// TwinCAT 3 PLC project TcMatrixTest
// Title: TcMatrix Unit Tests
// Company: Burks Engineering
// Author: Andrew Burks
// ProjectVersion: 0.0.0
// Description: Unit Tests for the TcMatrix Library
// ProgramVersion: 3.1.4023.0
// libraries:
//   Tc2_Standard, * (Beckhoff Automation GmbH)
//   Tc2_System, * (Beckhoff Automation GmbH)
//   Tc3_DynamicMemory, * (Beckhoff Automation GmbH)
//   Tc3_Module, * (Beckhoff Automation GmbH)
//   TcMatrix, * (Burks Engineering)
//   TcUnit,1.2.0.0,www.tcunit.org
// project tree:
//   / PlcTask.TcTTO
//   TESTs/ FB_CsvReadWrite_Test.TcPOU, FB_Array_Test.TcPOU, FB_MatrixElementProduct_Test.TcPOU, FB_MatrixDeterminate_Test.TcPOU, FB_MatrixGetMagicSquare_Test.TcPOU, FB_MatrixGrow_Test.TcPOU, FB_MatrixMatrixProduct_Test.TcPOU, FB_MatrixInvert_Test.TcPOU, FB_MatrixShrink_Test.TcPOU, FB_MatrixElementSum_Test.TcPOU, FB_MatrixSubMatrix_Test.TcPOU, FB_DynamicMatrix_Test.TcPOU, FB_MatrixTranspose_Test.TcPOU, FB_StaticMatrix_Test.TcPOU, FB_VectorCrossProduct_Test.TcPOU, PRG_TEST.TcPOU
//   Version/ Global_Version.TcGVL
// real-time tasks:
//   TASK PlcTask: cycle T#10ms, priority 20, ADS port 350

CONFIGURATION TcMatrixTest
    RESOURCE PLC ON TwinCAT3
        TASK PlcTask(INTERVAL := T#10ms, PRIORITY := 20);
        PROGRAM PRG_TEST WITH PlcTask : PRG_TEST;
    END_RESOURCE
END_CONFIGURATION

// ---- Version/Global_Version.TcGVL
{attribute 'TcGenerated'}
{attribute 'no-analysis'}
{attribute 'linkalways'}
// This function has been automatically generated from the project information.
VAR_GLOBAL CONSTANT
	{attribute 'const_non_replaced'}
	stLibVersion_TcMatrix_Unit_Tests : ST_LibVersion := (iMajor := 0, iMinor := 0, iBuild := 0, iRevision := 0, nFlags := 0, sVersion := '0.0.0');
END_VAR

// ---- TESTs/PRG_TEST.TcPOU
PROGRAM PRG_TEST
VAR
	fbDynamicMatrix : FB_DynamicMatrix_Test;
	fbArray: FB_Array_Test;
	fbMatrixGetMagicSquare : FB_MatrixGetMagicSquare_Test;
	fbMatrixSubmatrix : FB_MatrixSubMatrix_Test;
	fbMatrixGrow : FB_MatrixGrow_Test;
	fbMatrixShrink : FB_MatrixShrink_Test;
	fbMatrixElementSum : FB_MatrixElementSum_Test;
	fbMatrixElementProduct : FB_MatrixElementProduct_Test;
	fbMatrixDeterminate : FB_MatrixDeterminate_Test;
	fbMatrixMatrixProduct : FB_MatrixMatrixProduct_Test;
	fbVectorCrossProdcut : FB_VectorCrossProduct_Test;
	fbStaticMatrix : FB_StaticMatrix_Test;
	fbMatrixTranspose : FB_MatrixTranspose_Test;
	fbMatrixInvert : FB_MatrixInvert_Test;
	fbCsvReadWrite : FB_CsvReadWrite_Test;
END_VAR

TcUnit.RUN();

END_PROGRAM

// ---- TESTs/FB_DynamicMatrix_Test.TcPOU
FUNCTION_BLOCK FB_DynamicMatrix_Test EXTENDS FB_TestSuite
VAR_INPUT
END_VAR
VAR_OUTPUT
END_VAR
VAR
END_VAR

WhenInitiallyResizedExpectMemoryAllocated();
WhenResizedBiggerExpectMoreMemoryAllocated();
WhenResizedSmallerExpectLessMemoryAllocated();
WhenResizedToZeroExpectNoMemoryAllocated();

METHOD PRIVATE WhenInitiallyResizedExpectMemoryAllocated
VAR_INPUT
END_VAR

VAR
	M : DynamicMatrix;
	ResizeSuccess : BOOL;

END_VAR
TEST('WhenInitiallyResizedExpectMemoryAllocated');

// @TEST-RUN
ResizeSuccess := M.Resize(1,1,FALSE,TRUE);



// @TEST-ASSERT
AssertTrue(Condition :=ResizeSuccess,
	message := 'Error on valid initial resize');

	
TEST_FINISHED();
END_METHOD

METHOD PRIVATE WhenResizedBiggerExpectMoreMemoryAllocated
VAR_INPUT
END_VAR
VAR
	M : DynamicMatrix;
	InitialResizeSuccess : BOOL;
	SecondResizeSuccess : BOOL;

END_VAR
TEST('WhenResizedBiggerExpectMoreMemoryAllocated');

// @TEST-RUN
InitialResizeSuccess := M.Resize(1,1,FALSE,TRUE);
SecondResizeSuccess := M.Resize(2,2,FALSE,TRUE);


// @TEST-ASSERT
AssertTrue(Condition :=InitialResizeSuccess,
	message := 'Error on valid initial resize');
AssertTrue(Condition :=SecondResizeSuccess,
	message := 'Error on valid second resize');

	
TEST_FINISHED();
END_METHOD

METHOD PRIVATE WhenResizedSmallerExpectLessMemoryAllocated
VAR_INPUT
END_VAR
VAR
	M : DynamicMatrix;
	InitialResizeSuccess : BOOL;
	SecondResizeSuccess : BOOL;
	
END_VAR
TEST('WhenResizedSmallerExpectLessMemoryAllocated');

// @TEST-RUN
InitialResizeSuccess := M.Resize(2,2,FALSE,TRUE);
SecondResizeSuccess := M.Resize(1,1,FALSE,TRUE);

// @TEST-ASSERT
AssertTrue(Condition :=InitialResizeSuccess,
	message := 'Error on valid initial resize');
AssertTrue(Condition :=SecondResizeSuccess,
	message := 'Error on valid second resize');

	
TEST_FINISHED();
END_METHOD

METHOD PRIVATE WhenResizedToZeroExpectNoMemoryAllocated
VAR_INPUT
END_VAR
VAR
	M : DynamicMatrix;
	InitialResizeSuccess : BOOL;
	SecondResizeSuccess : BOOL;

END_VAR
TEST('WhenResizedToZeroExpectNoMemoryAllocated');

// @TEST-RUN
InitialResizeSuccess := M.Resize(1,1,FALSE,TRUE);
SecondResizeSuccess := M.Resize(0,0,FALSE,TRUE);


// @TEST-ASSERT
AssertTrue(Condition :=InitialResizeSuccess,
	message := 'Error on valid initial resize');
AssertTrue(Condition :=SecondResizeSuccess,
	message := 'Error on valid second resize');

	
TEST_FINISHED();
END_METHOD

END_FUNCTION_BLOCK

// ---- TESTs/FB_Array_Test.TcPOU
FUNCTION_BLOCK FB_Array_Test EXTENDS FB_TestSuite
VAR_INPUT
END_VAR
VAR_OUTPUT
END_VAR
VAR
END_VAR

WhenDynamicInitializedExpectValuesCopied();
WhenStaticInitializedExpectValuesCopied();
MarkdownExample1();

METHOD PRIVATE MarkdownExample1
VAR_INPUT
END_VAR
VAR
	M : Array2DStaticMatrix; //This instance is the matrix that the code will interact with
	M_Data : ARRAY[1..3,1..3] OF LREAL; //This array will act as the memory for the matrix
	V : Array2DStaticMatrix; //This instance is the initial column vector
	V_Data : ARRAY[1..3,1..1] OF LREAL := [1, 2, 3]; //This array will act as the memory for the initial column vector, prepopulated
	Res : Array2DStaticMatrix; //This instance is the resulting column vector
	Res_Data : ARRAY[1..3,1..1] OF LREAL := [1, 2, 3]; //This array will act as the memory for the resulting column vector
	success : BOOL; //records success or failure of the matrix multiplication
	equal : BOOL; //records success if the resulting vector is equal to the first
END_VAR
TEST('MarkdownExample1');

// @TEST-RUN
M(Data := M_Data); //Connect the memory to the matrix and initialize it
V(Data := V_Data); //Connect the memory to the initial column vector and initialize it (retaining declared values)
Res(Data := Res_Data); //Connect the memory to the resulting column vector and initialize it

M.FillTrapezoidal(Diagonal := 1, UpperRight := 0, LowerLeft := 0); //Transforms the matrix from all zeros into the identity matrix
success := Matrix_Product(M,V,Res); //perform the matrix multiplication
equal := V.IsEqual(Res); //the result of the multiplication should be equal to the initial value because of the identity matrix
	

// @TEST-ASSERT
AssertTrue(Condition :=success,
	message := 'Error on valid initial resize');
AssertTrue(Condition :=equal,
	message := 'Error on valid initial resize');
TEST_FINISHED();
END_METHOD

METHOD PRIVATE WhenDynamicInitializedExpectValuesCopied
VAR_INPUT
END_VAR
VAR
	A : ARRAY[1..3, 1..3] OF LREAL := [1,2,3,4,5,6,7,8,9];
	M : DynamicMatrix;
	
	InitSuccess : BOOL;
	
	ExpectedRank : UINT := 3;
	ExpectedVal : LREAL := 8.0; //expected at A[3,2] and M(2,1)
	
	MatrixRows : UINT;
	MatrixCols : UINT;
	ArrayVal : LREAL;
	MatrixVal : LREAL;

END_VAR
TEST('WhenDynamicInitializedExpectValuesCopied');

// @TEST-RUN
InitSuccess := M.InitArray2D(A);

MatrixRows := M.Rows;
MatrixCols := M.Cols;
ArrayVal := A[3,2];
MatrixVal := M.GetRC(2,1);


// @TEST-ASSERT
AssertTrue(Condition :=InitSuccess,
	message := 'Error on valid initial resize');
AssertEquals(Expected := ExpectedRank,
	Actual := MatrixRows,
	Message := 'Matrix row size not correct');
AssertEquals(Expected := ExpectedRank,
	Actual := MatrixCols,
	Message := 'Matrix col size not correct');
	
AssertEquals(Expected := ExpectedVal,
	Actual := ArrayVal,
	Message := 'Array content at [3,2] not correct');
	
AssertEquals(Expected := ExpectedVal,
	Actual := MatrixVal,
	Message := 'Matrix content at (2,1) not correct');
	
TEST_FINISHED();
END_METHOD

METHOD PRIVATE WhenStaticInitializedExpectValuesCopied
VAR_INPUT
END_VAR
VAR
	A : ARRAY[1..3, 1..3] OF LREAL := [1,2,3,4,5,6,7,8,9];
	M : Array2DStaticMatrix;
	
	ExpectedRank : UINT := 3;
	ExpectedVal : LREAL := 8.0; //expected at A[3,2] and M(2,1)
	
	MatrixRows : UINT;
	MatrixCols : UINT;
	ArrayVal : LREAL;
	MatrixVal : LREAL;

END_VAR
TEST('WhenStaticInitializedExpectValuesCopied');

// @TEST-RUN
M(Data := A);

MatrixRows := M.Rows;
MatrixCols := M.Cols;
ArrayVal := A[3,2];
MatrixVal := M.GetRC(2,1);


// @TEST-ASSERT
AssertEquals(Expected := ExpectedRank,
	Actual := MatrixRows,
	Message := 'Matrix row size not correct');
AssertEquals(Expected := ExpectedRank,
	Actual := MatrixCols,
	Message := 'Matrix col size not correct');
	
AssertEquals(Expected := ExpectedVal,
	Actual := ArrayVal,
	Message := 'Array content at [3,2] not correct');
	
AssertEquals(Expected := ExpectedVal,
	Actual := MatrixVal,
	Message := 'Matrix content at (2,1) not correct');
	
TEST_FINISHED();
END_METHOD

END_FUNCTION_BLOCK

// ---- TESTs/FB_MatrixGetMagicSquare_Test.TcPOU
FUNCTION_BLOCK FB_MatrixGetMagicSquare_Test EXTENDS FB_TestSuite
VAR_INPUT
END_VAR
VAR_OUTPUT
END_VAR
VAR
END_VAR

WhenCreatedExpectMagicProperties();

METHOD PRIVATE WhenCreatedExpectMagicProperties
VAR_INPUT
END_VAR
VAR
	M1 : DynamicMatrix;
	V : DynamicMatrix;
	Actual : LREAL;
	Expected : LREAL := 15;
	I : UINT;
END_VAR
TEST('WhenCreatedExpectMagicProperties');

// @TEST-RUN
M1.InitMagicSquare(3);//all rows and cols are 15
M1.LogData('3x3 Magic Square');

// @TEST-ASSERT
FOR I := 0 TO M1.Rows-1 DO
	//V.AsRowVector(M1,I); //cannot use, untested at this point
	Actual :=  M1.GetRC(I,0) + M1.GetRC(I,1) + M1.GetRC(I,2);//V.Sum; //cannot use, untested at this point
	AssertEquals(Expected,Actual,'Row is not the magic number');
END_FOR
FOR I := 0 TO M1.Cols-1 DO
	//V.AsRowVector(M1,I); //cannot use, untested at this point
	Actual :=  M1.GetRC(0,I) + M1.GetRC(1,I) + M1.GetRC(2,I);//V.Sum; //cannot use, untested at this point
	AssertEquals(Expected,Actual,'Col is not the magic number');
END_FOR

TEST_FINISHED();
END_METHOD

END_FUNCTION_BLOCK

// ---- TESTs/FB_MatrixSubMatrix_Test.TcPOU
{attribute 'reflection'}
FUNCTION_BLOCK FB_MatrixSubMatrix_Test EXTENDS FB_TestSuite
VAR_INPUT
END_VAR
VAR_OUTPUT
END_VAR
VAR
END_VAR

WhenCreatedExpectDataRetained();

METHOD PRIVATE WhenCreatedExpectDataRetained
VAR_INPUT
END_VAR
VAR
	M1 : DynamicMatrix;
	M2 : DynamicMatrix;
	Result : BOOL;
	
	Ri : UINT;
	Ci : UINT;
	
	Expected : LREAL;
	Actual : LREAL;
END_VAR
TEST('WhenCreatedExpectDataRetained');

// @TEST-RUN
M1.InitMagicSquare(5);
Result := M2.AsSubMatrix(M1,1,3,1,3);

// @TEST-ASSERT
AssertTrue(Result,'Main function call was not successful');

FOR Ri := 0 TO M2.Rows-1 DO
	FOR Ci := 0 TO M2.Cols-1 DO
		Expected := M1.GetRC(Ri+1,Ci+1);
		Actual := M2.GetRC(Ri,Ci);
		AssertEquals(Expected, Actual, 'Equivalent values are not equal after submatrix');
	END_FOR;
END_FOR

TEST_FINISHED();
END_METHOD

END_FUNCTION_BLOCK

// ---- TESTs/FB_MatrixGrow_Test.TcPOU
FUNCTION_BLOCK FB_MatrixGrow_Test EXTENDS FB_TestSuite
VAR_INPUT
END_VAR
VAR_OUTPUT
END_VAR
VAR
END_VAR

WhenEmptyExpectNoError();
WhenGrownExpectDataRetained();
WhenGrownExpectNewDataFilled();

METHOD PRIVATE WhenEmptyExpectNoError
VAR_INPUT
END_VAR
VAR
	M1 : DynamicMatrix;
	M2 : DynamicMatrix;
	Result : BOOL;
END_VAR
TEST('WhenEmptyExpectNoError');

// @TEST-RUN
M1.Init(0,0);
Result := M2.AsGrown(M1,0,0,0,0,0);

// @TEST-ASSERT
AssertTrue(Result,'Main function call was not successful');

TEST_FINISHED();
END_METHOD

METHOD PRIVATE WhenGrownExpectDataRetained
VAR_INPUT
END_VAR
VAR
	M1 : DynamicMatrix;
	M2 : DynamicMatrix;
	M3 : DynamicMatrix;
	Result : BOOL;
END_VAR
TEST('WhenGrownExpectDataRetained');

// @TEST-RUN
M1.InitMagicSquare(3);
Result := M2.AsGrown(M1,0,0,0,0,0);
M3.AsSubMatrix(M2,1,3,1,3);

// @TEST-ASSERT
AssertTrue(Result,'Main function call was not successful');
AssertTrue(M3.IsEqual(M1),'Old data was not retained');

TEST_FINISHED();
END_METHOD

METHOD PRIVATE WhenGrownExpectNewDataFilled
VAR_INPUT
END_VAR
VAR
	M1 : DynamicMatrix;
	M2 : DynamicMatrix;
	Result : BOOL;
END_VAR
TEST('WhenGrownExpectNewDataFilled');

// @TEST-RUN
M1.InitZeros(3,3);
Result := M2.AsGrown(M1,0,0,1,2,3);

// @TEST-ASSERT
AssertTrue(Result,'Main function call was not successful');
AssertTrue(M2.GetRC(0,0) = 1,'Diagonal data was not filled');
AssertTrue(M2.GetRC(0,1) = 2,'Row data was not filled');
AssertTrue(M2.GetRC(1,0) = 3,'Col data was not filled');

TEST_FINISHED();
END_METHOD

END_FUNCTION_BLOCK

// ---- TESTs/FB_MatrixShrink_Test.TcPOU
FUNCTION_BLOCK FB_MatrixShrink_Test EXTENDS FB_TestSuite
VAR_INPUT
END_VAR
VAR_OUTPUT
END_VAR
VAR
END_VAR

WhenEmptyExpectError();
WhenShrunkExpectDataRetained();

METHOD PRIVATE WhenEmptyExpectError
VAR_INPUT
END_VAR
VAR
	M1 : DynamicMatrix;
	M2 : DynamicMatrix;
	Result : BOOL;
END_VAR
TEST('WhenEmptyExpectError');

// @TEST-RUN
M1.InitZeros(1,1);
Result := M2.AsShrunk(M1,0,0);

// @TEST-ASSERT
AssertFalse(Result,'Main function call was unexpectedly successful');

TEST_FINISHED();
END_METHOD

METHOD PRIVATE WhenShrunkExpectDataRetained
VAR_INPUT
END_VAR
VAR
	M1 : DynamicMatrix;
	M2 : DynamicMatrix;
	M3 : DynamicMatrix;
	Result : BOOL;
END_VAR
TEST('WhenShrunkExpectDataRetained');

// @TEST-RUN
M1.InitMagicSquare(3);
Result := M2.AsShrunk(M1,0,0);
M3.AsSubMatrix(M1,1,2,1,2);

// @TEST-ASSERT
AssertTrue(Result,'Main function call was not successful');
AssertTrue(M3.IsEqual(M2),'Old data was not retained');

TEST_FINISHED();
END_METHOD

END_FUNCTION_BLOCK

// ---- TESTs/FB_MatrixElementSum_Test.TcPOU
FUNCTION_BLOCK FB_MatrixElementSum_Test EXTENDS FB_TestSuite
VAR_INPUT
END_VAR
VAR_OUTPUT
END_VAR
VAR
END_VAR

WhenDifferentExpectError();
WhenmatchingExpectResult();

METHOD PRIVATE WhenDifferentExpectError
VAR_INPUT
END_VAR
VAR
	M1 : DynamicMatrix;
	M2 : DynamicMatrix;
	M3 : DynamicMatrix;
	Result : BOOL;
END_VAR
TEST('WhenDifferentExpectError');

// @TEST-RUN
M1.InitMagicSquare(3);
M2.InitMagicSquare(5);
Result := M3.AsElementSum(M1,M2);

// @TEST-ASSERT
AssertFalse(Result,'Main function call was unexpectedly successful');

TEST_FINISHED();
END_METHOD

METHOD PRIVATE WhenMatchingExpectResult
VAR_INPUT
END_VAR
VAR
	M1 : DynamicMatrix;
	M2 : DynamicMatrix;
	M3 : DynamicMatrix;
	Result : BOOL;
END_VAR
TEST('WhenMatchingExpectResult');

// @TEST-RUN
M1.InitMagicSquare(3);
M2.InitMagicSquare(3);
Result := M3.AsElementSum(M1,M2);
M1.Scale(2);

// @TEST-ASSERT
AssertTrue(Result,'Main function call was not successful');
AssertTrue(M3.IsEqual(M1),'Data was successfully added');

TEST_FINISHED();
END_METHOD

END_FUNCTION_BLOCK

// ---- TESTs/FB_MatrixElementProduct_Test.TcPOU
FUNCTION_BLOCK FB_MatrixElementProduct_Test EXTENDS FB_TestSuite
VAR_INPUT
END_VAR
VAR_OUTPUT
END_VAR
VAR
END_VAR

WhenDifferentExpectError();
WhenmatchingExpectResult();

METHOD PRIVATE WhenDifferentExpectError
VAR_INPUT
END_VAR
VAR
	M1 : DynamicMatrix;
	M2 : DynamicMatrix;
	M3 : DynamicMatrix;
	Result : BOOL;
END_VAR
TEST('WhenDifferentExpectError');

// @TEST-RUN
M1.InitMagicSquare(3);
M2.InitMagicSquare(5);
Result := M3.AsElementProduct(M1,M2);

// @TEST-ASSERT
AssertFalse(Result,'Main function call was unexpectedly successful');

TEST_FINISHED();
END_METHOD

METHOD PRIVATE WhenMatchingExpectResult
VAR_INPUT
END_VAR
VAR
	M1 : DynamicMatrix;
	M2 : DynamicMatrix;
	M3 : DynamicMatrix;
	Result : BOOL;
END_VAR
TEST('WhenMatchingExpectResult');

// @TEST-RUN
M1.InitMagicSquare(3);
M2.InitMagicSquare(3);
Result := M3.AsElementProduct(M1,M2);
M1.Power(2);

// @TEST-ASSERT
AssertTrue(Result,'Main function call was not successful');
AssertTrue(M3.IsEqual(M1),'Data was successfully multiplied');

TEST_FINISHED();
END_METHOD

END_FUNCTION_BLOCK

// ---- TESTs/FB_MatrixDeterminate_Test.TcPOU
FUNCTION_BLOCK FB_MatrixDeterminate_Test EXTENDS FB_TestSuite
VAR_INPUT
END_VAR
VAR_OUTPUT
END_VAR
VAR
END_VAR

WhenNotSquareExpectError();
WhenMatchingExpectResult();

METHOD PRIVATE WhenMatchingExpectResult
VAR_INPUT
END_VAR
VAR
	M1 : DynamicMatrix;
	Result : BOOL;
	Actual : LREAL;
	Expected : LREAL := 360;
END_VAR
TEST('WhenMatchingExpectResult');

// @TEST-RUN
M1.InitMagicSquare(3);
Result := Matrix_DeterminateSquare(M := M1,Res => Actual);

// @TEST-ASSERT
AssertTrue(Result,'Main function call was not successful');
AssertEquals(Expected,Actual,'Determinate value was incorrect');

TEST_FINISHED();
END_METHOD

METHOD PRIVATE WhenNotSquareExpectError
VAR_INPUT
END_VAR
VAR
	M1 : DynamicMatrix;
	Result : BOOL;
	Actual : LREAL;
	Expected : LREAL := 0;
END_VAR
TEST('WhenNotSquareExpectError');

// @TEST-RUN
M1.InitTrapezoidal(2,3,1,1,1);
Result := Matrix_DeterminateSquare(M := M1,Res => Actual);

// @TEST-ASSERT
AssertFalse(Result,'Main function call was unexpectedly successful');
AssertEquals(Expected,Actual,'Determinate value was incorrect');

TEST_FINISHED();
END_METHOD

END_FUNCTION_BLOCK

// ---- TESTs/FB_MatrixMatrixProduct_Test.TcPOU
FUNCTION_BLOCK FB_MatrixMatrixProduct_Test EXTENDS FB_TestSuite
VAR_INPUT
END_VAR
VAR_OUTPUT
END_VAR
VAR
END_VAR

WhenColumnsExpectError();
WhenOppositeExpectScalar();
WhenOppositeExpectSquare();
WhenWithIdentityExpectSame();

METHOD PRIVATE WhenColumnsExpectError
VAR_INPUT
END_VAR
VAR
	V1 : DynamicMatrix;
	V2 : DynamicMatrix;
	M1 : DynamicMatrix;
	Result : BOOL;
END_VAR
TEST('WhenColumnsExpectError');

// @TEST-RUN
V1.InitVector(3,1,1);
V2.InitVector(3,1,1);
Result := M1.AsMatrixProduct(V1,V2);

// @TEST-ASSERT
AssertFalse(Result,'Main function call was unexpectedly successful');

TEST_FINISHED();
END_METHOD

METHOD PRIVATE WhenOppositeExpectScalar
VAR_INPUT
END_VAR
VAR
	V1 : DynamicMatrix;
	V2 : DynamicMatrix;
	M1 : DynamicMatrix;
	Result : BOOL;
END_VAR
TEST('WhenOppositeExpectScalar');

// @TEST-RUN
V1.InitVector(3,1,1);
V2.InitVector(3,1,1);
V1.Transpose();
Result := M1.AsMatrixProduct(V1,V2);

// @TEST-ASSERT
AssertTrue(Result,'Main function call was not successful');
AssertTrue(M1.Length = 1,'Result was not a scalar');
AssertTrue(M1.GetI(0) = V1.GetVectorDotProduct(V2),'Result was not the same as a dot product');

TEST_FINISHED();
END_METHOD

METHOD PRIVATE WhenOppositeExpectSquare
VAR_INPUT
END_VAR
VAR
	V1 : DynamicMatrix;
	V2 : DynamicMatrix;
	M1 : DynamicMatrix;
	Result : BOOL;
END_VAR
TEST('WhenOppositeExpectSquare');

// @TEST-RUN
V1.InitVector(3,1,1);
V2.InitVector(3,1,1);
V2.Transpose();
Result := M1.AsMatrixProduct(V1,V2);

// @TEST-ASSERT
AssertTrue(Result,'Main function call was not successful');
AssertTrue(M1.Length = 9 AND M1.IsSquare,'Result was not a 3x3 square');
AssertTrue(M1.Sum = 36,'Result values are incorrect');

TEST_FINISHED();
END_METHOD

METHOD PRIVATE WhenWithIdentityExpectSame
VAR_INPUT
END_VAR
VAR
	V1 : DynamicMatrix;
	MI : DynamicMatrix;
	M1 : DynamicMatrix;
	Result : BOOL;
END_VAR
TEST('WhenWithIdentityExpectSame');

// @TEST-RUN
V1.InitVector(3,1,1);
MI.InitIdentity(3);
Result := M1.AsMatrixProduct(MI,V1);

// @TEST-ASSERT
AssertTrue(Result,'Main function call was not successful');
AssertTrue(V1.IsEqual(M1),'Result was not the same');

TEST_FINISHED();
END_METHOD

END_FUNCTION_BLOCK

// ---- TESTs/FB_VectorCrossProduct_Test.TcPOU
FUNCTION_BLOCK FB_VectorCrossProduct_Test EXTENDS FB_TestSuite
VAR_INPUT
END_VAR
VAR_OUTPUT
END_VAR
VAR
END_VAR

WhenWrongSizeExpectError();
WhenMatchingSizeExpectResult();
WhenBackwardsExpectOppositeResult();

METHOD PRIVATE WhenBackwardsExpectOppositeResult
VAR_INPUT
END_VAR
VAR
	MV : DynamicMatrix;
	V1 : DynamicMatrix;
	V2 : DynamicMatrix;
	V3 : DynamicMatrix;
	Vs : ARRAY[0..1] OF POINTER TO MAtrix;
	M1 : DynamicMatrix;
	Result : BOOL;
END_VAR
TEST('WhenBackwardsExpectOppositeResult');

// @TEST-RUN
Vs[1] := ADR(V1);
Vs[0] := ADR(V2);

MV.InitIdentity(3);
V1.AsColVector(MV,0);
V2.AsColVector(MV,1);
V3.AsColVector(MV,2);
V3.Scale(-1);

Result := M1.AsVectorCrossProduct(Vs);

// @TEST-ASSERT
AssertTrue(Result,'Main function call was not successful');
AssertTrue(M1.IsEqual(V3),'Result is the correct vector');

TEST_FINISHED();
END_METHOD

METHOD PRIVATE WhenMatchingSizeExpectResult
VAR_INPUT
END_VAR
VAR
	MV : DynamicMatrix;
	V1 : DynamicMatrix;
	V2 : DynamicMatrix;
	V3 : DynamicMatrix;
	Vs : ARRAY[0..1] OF POINTER TO MAtrix;
	M1 : DynamicMatrix;
	Result : BOOL;
END_VAR
TEST('WhenMatchingSizeExpectResult');

// @TEST-RUN
Vs[0] := ADR(V1);
Vs[1] := ADR(V2);

MV.InitIdentity(3);
V1.AsColVector(MV,0);
V2.AsColVector(MV,1);
V3.AsColVector(MV,2);

Result := M1.AsVectorCrossProduct(Vs);

// @TEST-ASSERT
AssertTrue(Result,'Main function call was not successful');
AssertTrue(M1.IsEqual(V3),'Result is not the correct vector');

TEST_FINISHED();
END_METHOD

METHOD PRIVATE WhenWrongSizeExpectError
VAR_INPUT
END_VAR
VAR
	V1 : DynamicMatrix;
	V2 : DynamicMatrix;
	Vs : ARRAY [0..1] OF POINTER TO Matrix;
	M1 : DynamicMatrix;
	Result : BOOL;
END_VAR
TEST('WhenWrongSizeExpectError');

// @TEST-RUN
Vs[0] := ADR(V1);
Vs[1] := ADR(V2);

V1.InitVector(3,1,1);
V2.InitVector(4,1,1);

Result := Vector_CrossProduct(M1,Vs);

// @TEST-ASSERT
AssertFalse(Result,'Main function call was unexpectedly successful');

TEST_FINISHED();
END_METHOD

END_FUNCTION_BLOCK

// ---- TESTs/FB_StaticMatrix_Test.TcPOU
FUNCTION_BLOCK FB_StaticMatrix_Test EXTENDS FB_TestSuite
VAR_INPUT
END_VAR
VAR_OUTPUT
END_VAR
VAR
END_VAR

WhenCreatedExpectDataAssignable();

METHOD PRIVATE WhenCreatedExpectDataAssignable
VAR_INPUT
END_VAR
VAR
	M1 : ExternalStaticMatrix;
	M2 : DynamicMatrix;
	Data : ARRAY[0..8] OF LREAL;
	
	
END_VAR
TEST('WhenCreatedExpectDataAssignable');

// @TEST-RUN
M2.InitMagicSquare(3);
M1.Init(ADR(Data),3,3);
M1.FillFrom(M2);


// @TEST-ASSERT
AssertTrue(M1.IsEqual(M2),'Data was not all assigned');

TEST_FINISHED();
END_METHOD

END_FUNCTION_BLOCK

// ---- TESTs/FB_MatrixTranspose_Test.TcPOU
FUNCTION_BLOCK FB_MatrixTranspose_Test EXTENDS FB_TestSuite
VAR_INPUT
END_VAR
VAR_OUTPUT
END_VAR
VAR
END_VAR

WhenSquareExpectTranspose();
WhenDynamicRectangleExpectTranspose();
WhenStaticRectangleExpectTranspose();

METHOD PRIVATE WhenDynamicRectangleExpectTranspose
VAR_INPUT
END_VAR
VAR
	M1 : DynamicMatrix;
	M2 : DynamicMatrix;
	
	Result : BOOL;
END_VAR
TEST('WhenDynamicRectangleExpectTranspose');

// @TEST-RUN
M1.InitTrapezoidal(3,4,1,2,3);
Result := M1.Transpose();
M2.InitTrapezoidal(4,3,1,3,2);

// @TEST-ASSERT
AssertTrue(Result,'Main function call was not successful');

AssertTrue(M1.IsEqual(M2),'Data was not properly transposed');

TEST_FINISHED();
END_METHOD

METHOD PRIVATE WhenSquareExpectTranspose
VAR_INPUT
END_VAR
VAR
	M1 : DynamicMatrix;
	M2 : DynamicMatrix;
	
	Result : BOOL;
END_VAR
TEST('WhenSquareExpectTranspose');

// @TEST-RUN
M1.InitTrapezoidal(3,3,1,2,3);
Result := M1.Transpose();
M2.InitTrapezoidal(3,3,1,3,2);

// @TEST-ASSERT
AssertTrue(Result,'Main function call was not successful');

AssertTrue(M1.IsEqual(M2),'Data was not properly transposed');

TEST_FINISHED();
END_METHOD

METHOD PRIVATE WhenStaticRectangleExpectTranspose
VAR_INPUT
END_VAR
VAR
	M1 : ExternalStaticMatrix;
	M2 : DynamicMatrix;
	MT : TransposeMatrixAccessor;
	
	Data : ARRAY[0..11] OF LREAL;
	
	Result : BOOL;
END_VAR
TEST('WhenStaticRectangleExpectTranspose');

// @TEST-RUN
M1.Init(ADR(Data),3,4);
M1.FillTrapezoidal(1,2,3);
Mt := M1.GetTransposeMatrixAccessor();
M2.InitTrapezoidal(4,3,1,3,2);

// @TEST-ASSERT
AssertTrue(M2.IsEqual(MT),'Data was not properly transposed');

TEST_FINISHED();
END_METHOD

END_FUNCTION_BLOCK

// ---- TESTs/FB_MatrixInvert_Test.TcPOU
FUNCTION_BLOCK FB_MatrixInvert_Test EXTENDS FB_TestSuite
VAR_INPUT
END_VAR
VAR_OUTPUT
END_VAR
VAR
END_VAR

WhenIdentityExpectIdentity();
WhenSingularExpectError();
WhenSolvableExpectSolution();

METHOD PRIVATE WhenIdentityExpectIdentity
VAR_INPUT
END_VAR
VAR
	M1 : DynamicMatrix;
	M2 : DynamicMatrix;
	Result : BOOL;
END_VAR
TEST('WhenIdentityExpectIdentity');

// @TEST-RUN
M1.InitIdentity(3);
M2.InitIdentity(3);
Result := M2.InvertSquare(1E-9);

// @TEST-ASSERT
AssertTrue(Result,'Main function call was not successful');
AssertTrue(M1.IsNearlyEqual(M2,1E-6),'Result was not the same');

TEST_FINISHED();
END_METHOD

METHOD PRIVATE WhenSingularExpectError
VAR_INPUT
END_VAR
VAR
	M1 : DynamicMatrix;
	M2 : DynamicMatrix;
	Result : BOOL;
END_VAR
TEST('WhenSingularExpectError');

// @TEST-RUN
M1.InitTrapezoidal(3,3,1,1,1);
Result := M2.AsInverse(M1,1E-9);

// @TEST-ASSERT
AssertFalse(Result,'Main function call was surprisingly successful');

TEST_FINISHED();
END_METHOD

METHOD PRIVATE WhenSolvableExpectSolution
VAR_INPUT
END_VAR
VAR
	M1 : DynamicMatrix;
	M2 : DynamicMatrix;
	M3 : DynamicMatrix;
	M4 : DynamicMatrix;
	Result : BOOL;
END_VAR
TEST('WhenSolvableExpectSolution');

// @TEST-RUN
M1.InitIdentity(3);
M2.InitMagicSquare(3);
Result := M3.AsInverse(M2,1E-9);
M4.AsMatrixProduct(M2,M3);

// @TEST-ASSERT
AssertTrue(Result,'Main function call was not successful');
AssertTrue(M1.IsNearlyEqual(M4,1E-6),'Result was not a true inverse');

TEST_FINISHED();
END_METHOD

END_FUNCTION_BLOCK

// ---- TESTs/FB_CsvReadWrite_Test.TcPOU
FUNCTION_BLOCK FB_CsvReadWrite_Test EXTENDS FB_TestSuite
VAR_INPUT
END_VAR
VAR_OUTPUT
END_VAR
VAR
END_VAR

WhenWrittenThenReadExpectSame();

METHOD PRIVATE WhenWrittenThenReadExpectSame
VAR_INPUT
END_VAR
VAR_INST
	M1 : DynamicMatrix;
	M2 : DynamicMatrix;
	FilePath : T_MaxString := 'C:\ProgramData\TwinCAT PLC Control\Temporary Files\TcMatrix_CsvReadWriteTest_WhenWrittenThenReadExpectSame.csv';
	Writer : MatrixCsvWriter;
	Reader : MatrixCsvReader;
	
	step : UINT := 0;
	
	WriteError : BOOL;
	ReadError : BOOL;
END_VAR
VAR CONSTANT
	stepSetup : UINT := 0;
	stepWrite : UINT := 1;
	stepRead : UINT := 2;
	stepEvaluate : UINT := 3;
END_VAR
Writer(bExecute := step = stepWrite,
	M := M1,
	sPathname := FilePath,
	tTimeout := T#5S,
	pHeader := 0,
	cbHeaderLen := 0);
	
Reader(bExecute := step = stepRead,
	M := M2,
	sPathName := FilePath,
	tTimeout := T#5S,
	nHeaderLines := 0);

CASE step OF
	stepSetup:
		TEST('WhenWrittenThenReadExpectSame');
		M1.InitMagicSquare(25);
		M2.InitZeros(M1.Rows,M1.Cols);
		step := stepWrite;
		
	stepWrite:
		IF NOT Writer.bBusy THEN
			WriteError := Writer.bError;
			step := stepRead;
		END_IF
		
	stepRead:
		IF NOT Reader.bBusy THEN
			ReadError := Reader.bError;
			step := stepEvaluate;
		END_IF
		
	stepEvaluate:
		AssertTrue(NOT (WriteError), 'Writer error');
		AssertTrue(NOT  (ReadError), 'Reader error');
		AssertTrue(M1.IsEqual(M2), 'Data not transferred');
		TEST_FINISHED();
END_CASE
END_METHOD

END_FUNCTION_BLOCK
